// TIA Portal V20 export
TYPE "typeEm7Commands"
// stored: Access Published, Namespace Unit1
   STRUCT
      jobinterface { ExternalWritable := 'False'} : "Unit1.typeEm7CommandsJobInterface";
   END_STRUCT;
END_TYPE
